// TIA Portal V19 export
TYPE "C302_VAR_LKM_TYPIC"
   STRUCT
      MWA { ExternalAccessible := 'False'; ExternalVisible := 'False'; ExternalWritable := 'False'} : USInt;   // Meetwaarde (uitgemiddelde k-waarde)
      POS { ExternalAccessible := 'False'; ExternalVisible := 'False'; ExternalWritable := 'False'} : USInt;   // Lengtepositie van de luchtkwaliteitsmeter in de verkeerskoker
      VAR_ROOK { ExternalAccessible := 'False'; ExternalVisible := 'False'; ExternalWritable := 'False'} : USInt;   // Rookdetectie
      OBS { ExternalAccessible := 'False'; ExternalVisible := 'False'; ExternalWritable := 'False'} : USInt;   // Observeerbaarheid
      NUM_VOOR { ExternalAccessible := 'False'; ExternalVisible := 'False'; ExternalWritable := 'False'} : Int;   // Nummer van de voorafgaande luchtkwaliteitsmeter
      NUM_NA { ExternalAccessible := 'False'; ExternalVisible := 'False'; ExternalWritable := 'False'} : Int;   // Nummer van de volgende luchtkwaliteitsmeter
   END_STRUCT;
END_TYPE
